Universal Robots PolyScope program: letra_A.urp

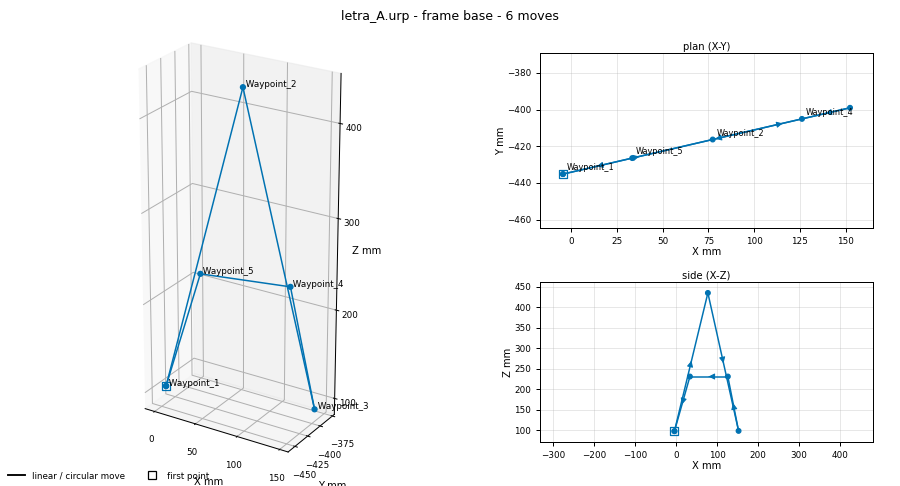
[picture p0: tool path of letra_A.urp in frame base, 6 of 6 moves have a stored position in this frame; points joined in program order, loops and branches not executed]
Program letra_A (installation=default directory=/ursim/programs createdIn=3.15.8.106339 lastSavedIn=3.15.8.106339 robotSerialNumber=2018359999)
Calibrated DH parameters: a=[0, -0.425, -0.39225, 0, 0, 0]; d=[0.089159, 0, 0, 0.10915, 0.09465, 0.0823]; alpha=[1.570796, 0, 0, 1.570796, -1.570796, 0]; deltaTheta=[0, 0, 0, 0, 0, 0]
Robot Program (runOnlyOnce=false)
  Popup Message (haltProgram=false message=Simulando letra A inputType=Text)
  MoveL speed 250 mm/s, acceleration 1200 mm/s^2 (useActiveTCP=true) feature=Base
    Waypoint Waypoint_1: TCP in base x=-4.389 y=-435.209 z=97.379 mm, rx=-0.0012 ry=3.1163 rz=0.0389 rad; joints [-76.392, -103.939, -130.798, -36.316, 91.732, 13.547] deg
    Waypoint Waypoint_2: TCP in base x=77.362 y=-416.323 z=435.326 mm, rx=-0.0012 ry=3.1163 rz=0.0389 rad; joints [-64.919, -79.715, -98.622, -92.35, 91.907, 25.025] deg
    Waypoint Waypoint_3: TCP in base x=152.363 y=-398.996 z=98.14 mm, rx=-0.0012 ry=3.1163 rz=0.0389 rad; joints [-54.691, -103.037, -132.205, -35.096, 91.999, 35.258] deg
    Waypoint Waypoint_4: TCP in base x=126.115 y=-405.06 z=231.01 mm, rx=-0.0012 ry=3.1163 rz=0.0389 rad; joints [-58.193, -87.176, -123.416, -59.867, 91.974, 31.754] deg
    Waypoint Waypoint_5: TCP in base x=33.429 y=-426.472 z=231.01 mm, rx=-0.0012 ry=3.1163 rz=0.0389 rad; joints [-71.098, -87.704, -122.798, -60.387, 91.822, 18.843] deg
    Waypoint Waypoint_1: TCP in base x=-4.389 y=-435.209 z=97.379 mm, rx=-0.0012 ry=3.1163 rz=0.0389 rad; joints [-76.392, -103.939, -130.798, -36.316, 91.732, 13.547] deg
